// TIA Portal V19 export
VAR_GLOBAL   // PLC tag table "LB302"
   LB302_ScaricoSemilavorati_SX_Pb_Aux1 AT %I251.5 : Bool;   // 344SH1
   LB302_ScaricoSemilavorati_SX_Pb_Aux2 AT %I251.6 : Bool;   // 344SH2
   LB302_ScaricoSemilavorati_SX_Lp_Aux1 AT %Q251.1 : Bool;   // 344SH1
   LB302_ScaricoSemilavorati_SX_Lp_Aux2 AT %Q251.2 : Bool;   // 344SH2
END_VAR
